// TIA Portal V19 export
TYPE "PositioningMachine_Alr"
// stored: Access Published
   STRUCT
      AxisNotInOperation : Bool;
      BrakeTimeOut : Bool;
      AxisTorqueLim : Struct
         Error : Bool;
         ErrorId : Word;
      END_STRUCT;
      Ax : "TAx_Alarms";
      Fan_M : "MotorAlr";
   END_STRUCT;
END_TYPE
